{attribute 'TcGenerated'}
{attribute 'no-analysis'}
{attribute 'linkalways'}
// This function has been automatically generated from the project information.
VAR_GLOBAL CONSTANT
	{attribute 'const_non_replaced'}
	stLibVersion_Math : ST_LibVersion := (iMajor := 0, iMinor := 0, iBuild := 2, iRevision := 0, nFlags := 0, sVersion := '0.0.2');
END_VAR

(* stored: Version 1.1.0.1, ProductVersion 3.1.4024.15
   GVL Global_Version: Id {55875edb-9b5e-0348-2d52-8e23a9b03de2} *)
